PROGRAM MAIN
VAR
	fbSupervisor	: FB_AGVSupervisor(sIPaddr := '127.0.0.1', nPort := 2000);
END_VAR


fbSupervisor();

END_PROGRAM

(* stored: Version 1.1.0.1, ProductVersion 3.1.4026.13
   POU MAIN: Id {3630ccad-c9cd-4213-8e6b-1c2fc4e308ce}, SpecialFunc None *)
